ABB RobotStudio station: cacona.rsstnx

Station Project1 (saved by RobotStudio 25.5.11605.0)
Controller IRB140_6_81
  mechanical unit ROB_1: IRB140_6_81_C_03, 6 joints, base frame (0, 0, 0) mm
Layout (positions relative to the parent item):
  - IRB140_6_81_C_03 [mechanism, from %ABB.RobotStudio.Models.IRB140%\IRB140_6_81_C_G_03.rslib] at (0, 0, 0) mm; joint values [0.4637, 0.408, -0.2217, -0.266, 0.9489, 0.5713] (rad or m)
Targets, tools, work objects and paths stored in the station, written as RAPID:
! task T_ROB1
MODULE Module1
  CONST robtarget Target_30:=[[506.291651246,0,679.5],[0.5,0,0.866025404,0],[0,0,0,0],[9E+09,9E+09,9E+09,9E+09,9E+09,9E+09]];
  PROC Path_10()
    MoveL Target_10_2,v500,z50,tool0\WObj:=wobj0;
    MoveL Target_10,v7000,z60,tool0\WObj:=wobj0;
    MoveL Target_20,v7000,z60,tool0\WObj:=wobj0;
    MoveL Target_10_4,v7000,z50,tool0\WObj:=wobj0;
    MoveL Target_30,v500,z50,tool0\WObj:=wobj0;
  ENDPROC
ENDMODULE

